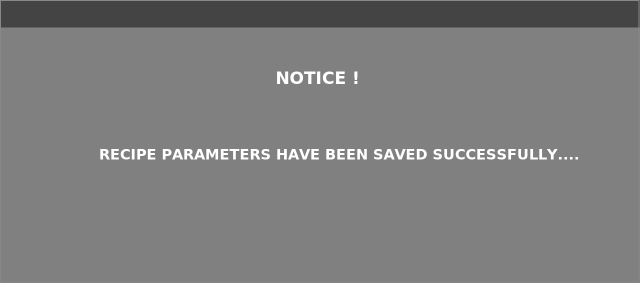
VISUALIZATION Popup_Parameter_Saved  // 640x283
    Rectangle (0,0 640x283)
    Rectangle (1,0 639x27)
    Label (262,66 101x24), "NOTICE !"
    Label (96,100 516x109), "RECIPE PARAMETERS HAVE BEEN SAVED SUCCESSFULLY...."
END_VISUALIZATION

(* stored: Version 1.1.0.1, ProductVersion 3.1.4024.12
   Visu Popup_Parameter_Saved: Id {103823d6-3d76-4a61-8748-1f2a200483f7} *)
